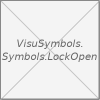
VISUALIZATION LoginButton  // 100x100
    Ellipse (0,0 100x100)
    Image (0,0 100x100), image: VisuSymbols.Symbols.Lock
        OnMouseDown: VisuUserMgmt Type=Login
    Ellipse (0,0 100x100)
    Image (0,0 100x100), image: VisuSymbols.Symbols.LockOpen
        OnMouseDown: VisuUserMgmt Type=Logout
END_VISUALIZATION

(* stored: Version 1.1.0.1, ProductVersion 3.1.4024.11
   Visu LoginButton: Id {4c6f2011-4174-4728-bad5-58f3738dbe64} *)
